# EPICS alarm handler configuration: alh_files/mgnt_li21_ycor.alhConfig
GROUP NULL YCOR:LI21:MG01
$ALIAS YCOR
$GUIDANCE
LI21 YCOR magnets
   Group Name: YCOR:LI21:MG01
   Summary PV:  YCOR:LI21:MG01:STATSUMY
$END

GROUP YCOR:LI21:MG01  YCOR:LI21:203
CHANNEL     YCOR:LI21:203         YCOR:LI21:203:STATMSG    -----
   $FORCEPV YCOR:LI21:203:STATMSGSV -DATL 1 0

GROUP YCOR:LI21:MG01  YCOR:LI21:303
CHANNEL     YCOR:LI21:303         YCOR:LI21:303:STATMSG    -----
   $FORCEPV YCOR:LI21:303:STATMSGSV -DATL 1 0

TD11 here!
GROUP YCOR:LI21:MG01  YCOR:LI21:403
CHANNEL     YCOR:LI21:403         YCOR:LI21:403:STATMSG    -----
   $FORCEPV YCOR:LI21:403:STATMSGSV -DATL 1 0

GROUP YCOR:LI21:MG01  YCOR:LI21:503
CHANNEL     YCOR:LI21:503         YCOR:LI21:503:STATMSG    -----
   $FORCEPV YCOR:LI21:503:STATMSGSV -DATL 1 0

GROUP YCOR:LI21:MG01  YCOR:LI21:603
CHANNEL     YCOR:LI21:603         YCOR:LI21:603:STATMSG    -----
   $FORCEPV YCOR:LI21:603:STATMSGSV -DATL 1 0

GROUP YCOR:LI21:MG01  YCOR:LI21:703
CHANNEL     YCOR:LI21:703         YCOR:LI21:703:STATMSG    -----
   $FORCEPV YCOR:LI21:703:STATMSGSV -DATL 1 0

GROUP YCOR:LI21:MG01  YCOR:LI21:803
CHANNEL     YCOR:LI21:803         YCOR:LI21:803:STATMSG    -----
   $FORCEPV YCOR:LI21:803:STATMSGSV -DATL 1 0

GROUP YCOR:LI21:MG01  YCOR:LI21:900
CHANNEL     YCOR:LI21:900         YCOR:LI21:900:STATMSG    -----
   $FORCEPV YCOR:LI21:900:STATMSGSV -DATL 1 0
